// TIA Portal V17 export
// export: Created 2023-02-14T02:49:50.9142998Z, ExportSetting WithDefaults, DisplayName Totally Integrated Automation Portal, DisplayVersion V17, DisplayName TIA Portal Openness, DisplayVersion V17, DisplayName TIA Portal Teamcenter Gateway, DisplayVersion V17, DisplayName TIA Portal Version Control Interface, DisplayVersion V17, DisplayName SINAMICS Startdrive Advanced, DisplayVersion V17, DisplayName SINAMICS Startdrive G130, G150, S120, S150, SINAMICS MV, S210, DisplayVersion V17, DisplayName SINAMICS Startdrive G110M, G120, G120C, G120D, G120P, G115D, DisplayVersion V17, DisplayName STEP 7 Professional, DisplayVersion V17, DisplayName STEP 7 Safety, DisplayVersion V17, DisplayName WinCC Professional, DisplayVersion V17
DATA_BLOCK "T-10.01_DB"   // DB360
VERSION : 0.1
// stored: AutoNumber false, DBAccessibleFromOPCUA true, DBAccessibleFromWebserver true, InstanceOfName BFT_Type5, InstanceOfType FB
"BFT_Type5"
   // VAR_INPUT
   //    "IN_FBAV.01" : Bool;
   //    "IN_FBAV.02" : Bool;
   //    "IN_FBAV.03" : Bool;
   //    "IN_FBSV.01" : Bool;
   //    IN_LT01 : Real;
   //    "IN_FBP.01" : Bool;
   //    "IN_P.01-Speed" : Real;
   //    DosePumpSpeed : Real;
   //    "DoseON-OFF" : Bool;
   //    "DosePumpON-OFF" : Bool;
   //    CIPPulse : Bool;
   //    CIP_Supply_ON : Bool;
   //    CIP_Busy : Bool;
   //    LineTrf_OK : Bool;
   //    LineFlush_OK : Bool;
   //    LCS_Start : Bool;
   //    LCS_Stop : Bool;
   // END_VAR
   // VAR_OUTPUT
   //    "OUT_AV.01" : Bool;
   //    "OUT_AV.02" : Bool;
   //    "OUT_AV.03" : Bool;
   //    "OUT_AV.06" : Bool;
   //    "OUT_P.01" : Bool;
   //    "OUT_P.01-Speed" : Real;
   //    "OUT_SV.01" : Bool;
   //    OUT_CIPTank_AVOpen : Bool;
   // END_VAR
   // VAR
   //    Cmd { ExternalVisible := 'False'} : Struct
   //       Inload { ExternalVisible := 'False'} : Bool;
   //       RaadyForMix { ExternalVisible := 'False'} : Bool;
   //       Tank_CIP_Req { ExternalVisible := 'False'} : Bool;
   //       Flush_Select { ExternalVisible := 'False'} : Byte;
   //       Flushing { ExternalVisible := 'False'} : Bool;
   //    END_STRUCT;
   //    Param { ExternalVisible := 'False'} : Struct
   //       SP_Level_LL { ExternalVisible := 'False'} : Real;
   //       SP_Level_ML { ExternalVisible := 'False'} : Real;
   //       SP_Level_HL { ExternalVisible := 'False'} : Real;
   //       L_Hi_Lim { ExternalVisible := 'False'} : Real;
   //       L_Lo_Lim { ExternalVisible := 'False'} : Real;
   //       L_Hys { ExternalVisible := 'False'} : Real;
   //       FlushingTime { ExternalVisible := 'False'} : Time;
   //       CIP_Trf_SP_Speed { ExternalVisible := 'False'} : Real;
   //       CIP_Ret_ON_SP { ExternalVisible := 'False'} : Real;
   //       CIP_Ret_OFF_SP { ExternalVisible := 'False'} : Real;
   //    END_STRUCT;
   //    State { ExternalVisible := 'False'} : Struct
   //       Tank_inloading { ExternalVisible := 'False'} : Bool;
   //       Tank_inRawDose { ExternalVisible := 'False'} : Bool;
   //       Tank_inCIP { ExternalVisible := 'False'} : Bool;
   //       Line_inCIP { ExternalVisible := 'False'} : Bool;
   //       Flushing { ExternalVisible := 'False'} : Bool;
   //       Tank_LL { ExternalVisible := 'False'} : Bool;
   //       Tank_ML { ExternalVisible := 'False'} : Bool;
   //       Tank_HL { ExternalVisible := 'False'} : Bool;
   //       Inload_Enable { ExternalVisible := 'False'} : Bool;
   //       Tank_CIP_Enable { ExternalVisible := 'False'} : Bool;
   //       Line_CIP_Enable { ExternalVisible := 'False'} : Bool;
   //       Flushing_Enable { ExternalVisible := 'False'} : Bool;
   //       Flush_selected { ExternalVisible := 'False'} : Byte;
   //       CIP_Request_OK { ExternalVisible := 'False'} : Bool;
   //       CIP_ReturnON { ExternalVisible := 'False'} : Bool;
   //       Ready_For_Transfer { ExternalVisible := 'False'} : Bool;
   //       Ready_For_Transfer_EN { ExternalVisible := 'False'} : Bool;
   //       Transfer_to_Blend { ExternalVisible := 'False'} : Bool;
   //       Status { ExternalVisible := 'False'} : Int;
   //    END_STRUCT;
   //    alwaysON : Bool;
   //    L_Hys_Abs : Real;
   //    Hys_Level_HL : Real;
   //    Hys_Level_ML : Real;
   //    Hys_Level_LL : Real;
   //    r : Struct
   //       PosE1 : Bool;
   //       PosE2 : Bool;
   //       PosE3 : Bool;
   //       PosE4 : Bool;
   //       PosE5 : Bool;
   //       PosE6 : Bool;
   //       PosE7 : Bool;
   //       PosE8 : Bool;
   //       PosE9 : Bool;
   //       PosE10 : Bool;
   //       PosE11 : Bool;
   //       PosE12 : Bool;
   //       PosE13 : Bool;
   //       PosE14 : Bool;
   //       PosE15 : Bool;
   //       PosE16 : Bool;
   //       PosE17 : Bool;
   //       PosE18 : Bool;
   //       PosE19 : Bool;
   //       PosE20 : Bool;
   //       PosE21 : Bool;
   //       PosE22 : Bool;
   //       PosE23 : Bool;
   //       PosE24 : Bool;
   //       PosE25 : Bool;
   //       PosE26 : Bool;
   //       PosE27 : Bool;
   //       PosE28 : Bool;
   //       PosE29 : Bool;
   //       PosE30 : Bool;
   //       PosE31 : Bool;
   //       PosE32 : Bool;
   //    END_STRUCT;
   //    Actuator : Struct
   //       AV_Outlet : Bool;
   //       TransferPump : Bool;
   //       FlushPump : Bool;
   //       CV_Steam : Bool;
   //       Pump : Bool;
   //       Agitator_level : Bool;
   //       LCS_OnOff : Bool;
   //    END_STRUCT;
   //    FlushingTim : TON_TIME;
   // END_VAR
BEGIN
END_DATA_BLOCK
